PROGRAM Main_Send
VAR	
	Done		: BOOL;
	New_Data	: BOOL;
	New_IMU		: BOOL;
	Sent		: BOOL;
	Saved		: BOOL;
	Sent_Data	: BOOL;
	Sent_IMU	: BOOL;
	Saved_Data	: BOOL;
	Saved_IMU	: BOOL;
	
	nState		: INT;

END_VAR

(* get data from database *)
Get_Data();
Get_IMU();

New_Data := Get_Data.Done;
New_IMU := Get_IMU.Done;
 
IF New_Data AND New_IMU THEN
	IF NOT Sent THEN
		(* send data to aws iot core *)
		Send();
		
		IF Send.Published_Data AND Send.Published_IMU THEN
			Sent	:= TRUE;
		END_IF	
		
	ELSE
		IF Save_Data.Done AND Save_IMU.Done THEN
			Saved := TRUE;
		END_IF	
		
	END_IF
	
ELSE
	Sent	:= FALSE;
	Saved 	:= FALSE;
	
END_IF

Save_Data();	
Save_IMU();

END_PROGRAM

(* stored: Version 1.1.0.1, ProductVersion 3.1.4024.6
   POU Main_Send: Id {f159ed40-cca9-4e3d-ac6a-ec5e9cf1af8e}, SpecialFunc None *)
